FUNCTION_BLOCK FB_System_BSp_Stellwertscheck
VAR_INPUT
	Stellwert	: ST_System_BSp_Stellwert;
	Zustand		: ST_System_BSp_Zustand;
END_VAR
VAR_OUTPUT
END_VAR
VAR
	Timer1		: TON;
END_VAR

(* überprüft, dass eine bestimmte Zeitperiode (Einschaltperiode_Max) vergangen ist, bis sich eine Pumpe wieder einschalten darf *)
Timer1(	IN := Zustand.Betrieb_Soll = FALSE AND Zustand.Stoerung = TRUE,
		PT := Stellwert.Einschaltperiode_Max,
		Q => Stellwert.Einschalten
);

END_FUNCTION_BLOCK

(* stored: Version 1.1.0.1, ProductVersion 3.1.4024.9
   POU FB_System_BSp_Stellwertscheck: Id {411a7999-b45d-4f72-9ac7-5bccf7a34d6f}, SpecialFunc None *)
